// TIA Portal project "Cement Mixing Project-Vinit" (V18)

(* hardware
DEVICE "S7-1200 station_1"  S7-1200 Station
   slot 0: "Rack_0"  S7-1200 Rack  Rack  V1.0
   slot 1: "PLC_1"  CPU 1212C AC/DC/Rly  6ES7 212-1BE40-0XB0  V4.6
*)

// ===== PLC "PLC_1"  CPU 1212C AC/DC/Rly =====

VAR_GLOBAL   // PLC tag table "Default tag table"
   "Flow Meter A" AT %I0.0 : Bool;
   "Valve A" AT %Q0.0 : Bool;
   "Flow Meter B" AT %I0.1 : Bool;
   "Valve B" AT %Q0.1 : Bool;
   "Mixing Motor" AT %Q0.3 : Bool;
   "Valve C" AT %Q0.2 : Bool;
   "LL Sensor" AT %I0.2 : Bool;
   "Start" AT %I0.3 : Bool;
   "Stop" AT %I0.4 : Bool;
   "Emergency_Stop" AT %I0.5 : Bool;
   "Emergency Stop Bit" AT %M0.0 : Bool;
   "Process_start" AT %M0.1 : Bool;
END_VAR

// folder: System blocks/Program resources

DATA_BLOCK "IEC_Counter_0_DB"   // DB1
{ S7_Optimized_Access := 'TRUE' }
AUTHOR : Simatic
FAMILY : IEC
NAME : CNTR
VERSION : 1.0
// stored: InstanceOfName IEC_COUNTER
"IEC_COUNTER"
BEGIN
END_DATA_BLOCK

DATA_BLOCK "IEC_Counter_0_DB_2"   // DB3
{ S7_Optimized_Access := 'TRUE' }
AUTHOR : Simatic
FAMILY : IEC
NAME : CNTR
VERSION : 1.0
// stored: InstanceOfName IEC_COUNTER
"IEC_COUNTER"
BEGIN
END_DATA_BLOCK

DATA_BLOCK "IEC_Timer_0_DB_2"   // DB4
{ S7_Optimized_Access := 'TRUE' }
AUTHOR : Simatic
FAMILY : IEC
NAME : IEC_TMR
VERSION : 1.0
// stored: InstanceOfName IEC_TIMER
"IEC_TIMER"
BEGIN
END_DATA_BLOCK

// folder: (top level)

ORGANIZATION_BLOCK "Main"   // OB1, LAD, ProgramCycle
TITLE = "Main Program Sweep (Cycle)"
{ S7_Optimized_Access := 'TRUE' }
VERSION : 0.1
   VAR_INPUT
      Initial_Call : Bool;   // Initial call of this OB
      Remanence : Bool;   // =True, if remanent data are available
   END_VAR
   VAR_TEMP   // added for the SCL form of the ladder/FBD networks
      _w1 : Bool;
   END_VAR
BEGIN

REGION Network 1: Start, Stop & Emergency Button
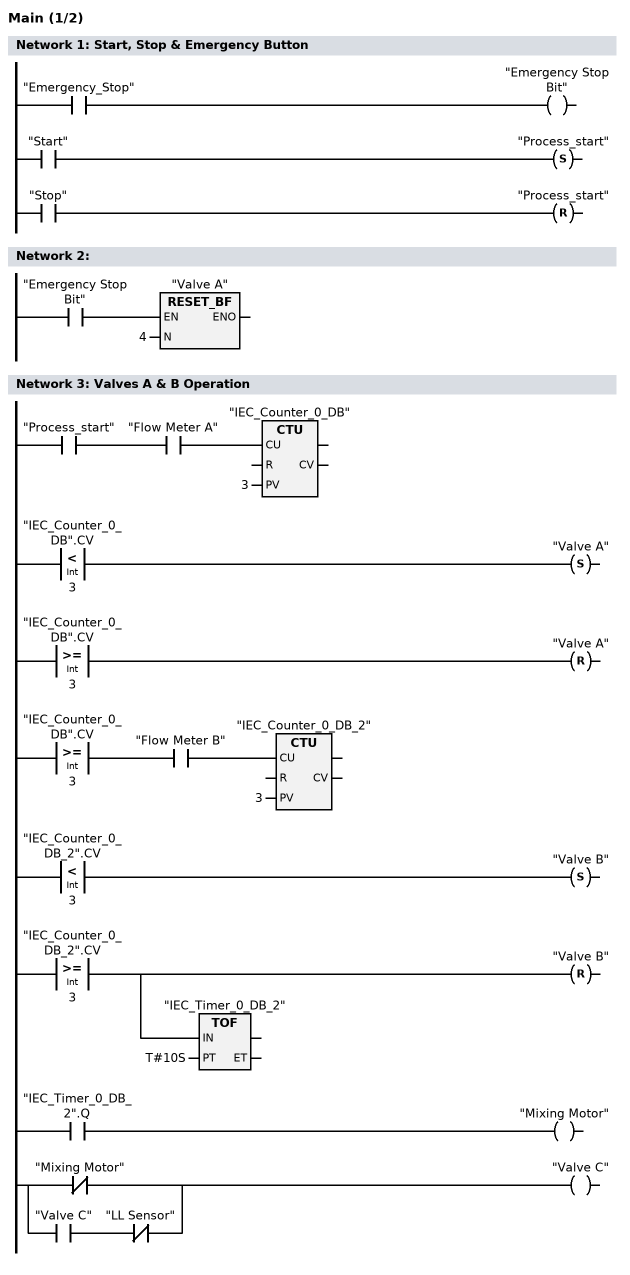
   RUNG wire#powerrail
      Contact( "Emergency_Stop" )
      Coil( "Emergency Stop Bit" )
   END_RUNG
   RUNG wire#powerrail
      Contact( "Start" )
      S_Coil( "Process_start" )
   END_RUNG
   RUNG wire#powerrail
      Contact( "Stop" )
      R_Coil( "Process_start" )
   END_RUNG
   // the same network as SCL:
   "Emergency Stop Bit" := "Emergency_Stop";
   IF "Start" THEN "Process_start" := TRUE; END_IF;
   IF "Stop" THEN "Process_start" := FALSE; END_IF;
END_REGION

REGION Network 2
   // no SCL statement known for RBitfield: written as a call
   IF "Emergency Stop Bit" THEN RESET_BF(operand := "Valve A", n := 4); END_IF;
END_REGION

REGION Network 3: Valves A & B Operation
   "IEC_Counter_0_DB".CTU(CU := "Process_start" AND "Flow Meter A", PV := 3);
   IF "IEC_Counter_0_DB".CV < 3 THEN "Valve A" := TRUE; END_IF;
   IF "IEC_Counter_0_DB".CV >= 3 THEN "Valve A" := FALSE; END_IF;
   "IEC_Counter_0_DB_2".CTU(CU := ("IEC_Counter_0_DB".CV >= 3) AND "Flow Meter B", PV := 3);
   IF "IEC_Counter_0_DB_2".CV < 3 THEN "Valve B" := TRUE; END_IF;
   #_w1 := "IEC_Counter_0_DB_2".CV >= 3;
   IF #_w1 THEN "Valve B" := FALSE; END_IF;
   "IEC_Timer_0_DB_2".TOF(IN := #_w1, PT := T#10S);
   "Mixing Motor" := "IEC_Timer_0_DB_2".Q;
   "Valve C" := NOT "Mixing Motor" OR ("Valve C" AND NOT "LL Sensor");
END_REGION

REGION Network 4: Mixer Operation
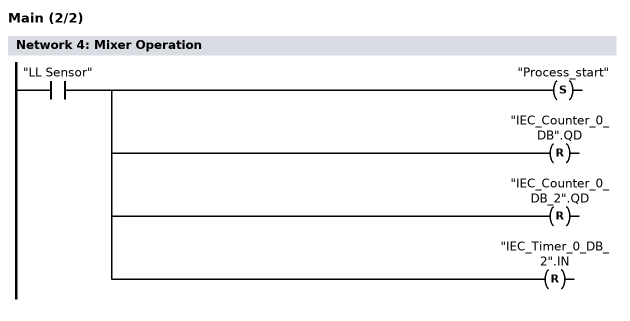
   RUNG wire#powerrail
      Contact( "LL Sensor" )
      wire#w1
      S_Coil( "Process_start" )
   END_RUNG
   RUNG wire#w1
      R_Coil( "IEC_Counter_0_DB".QD )
   END_RUNG
   RUNG wire#w1
      R_Coil( "IEC_Counter_0_DB_2".QD )
   END_RUNG
   RUNG wire#w1
      R_Coil( "IEC_Timer_0_DB_2".IN )
   END_RUNG
   // the same network as SCL:
   IF "LL Sensor" THEN
       "Process_start" := TRUE;
       "IEC_Counter_0_DB".QD := FALSE;
       "IEC_Counter_0_DB_2".QD := FALSE;
       "IEC_Timer_0_DB_2".IN := FALSE;
   END_IF;
END_REGION
END_ORGANIZATION_BLOCK